// SIMATIC S7-200 project (STEP 7-Micro/WIN), CPU 224 REL 02.01

ORGANIZATION_BLOCK MAIN:OB1
TITLE=PROGRAM COMMENTS
BEGIN
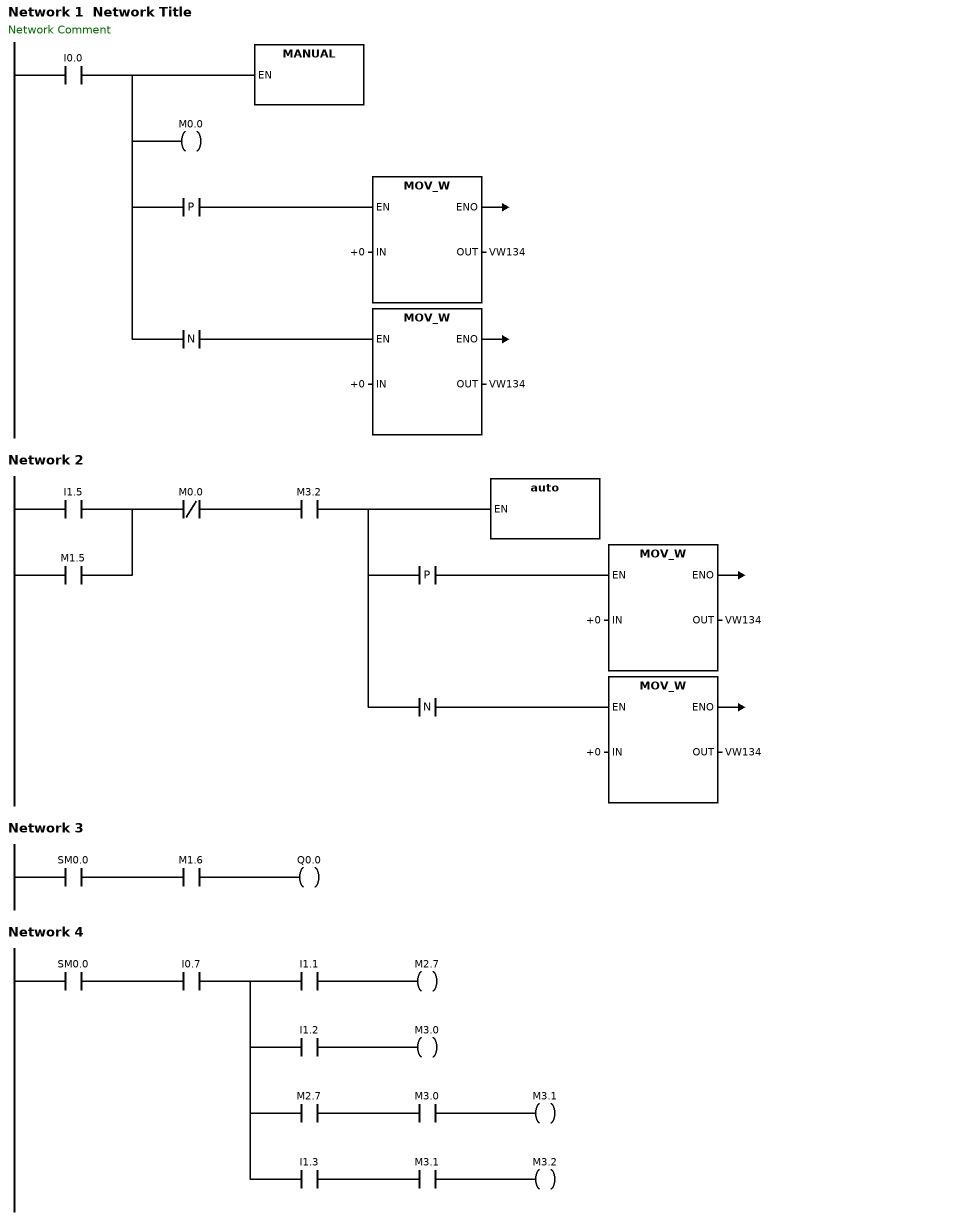
Network 1 // Network Title
// Network Comment
LD     I0.0
LPS
CALL   MANUAL:SBR0
=      M0.0
EU
MOVW   +0, VW134
LPP
ED
MOVW   +0, VW134
Network 2
LD     I1.5
O      M1.5
AN     M0.0
A      M3.2
LPS
CALL   auto:SBR1
EU
MOVW   +0, VW134
LPP
ED
MOVW   +0, VW134
Network 3
LD     SM0.0
A      M1.6
=      Q0.0
Network 4
LD     SM0.0
A      I0.7
LPS
A      I1.1
=      M2.7
LRD
A      I1.2
=      M3.0
LRD
A      M2.7
A      M3.0
=      M3.1
LPP
A      I1.3
A      M3.1
=      M3.2
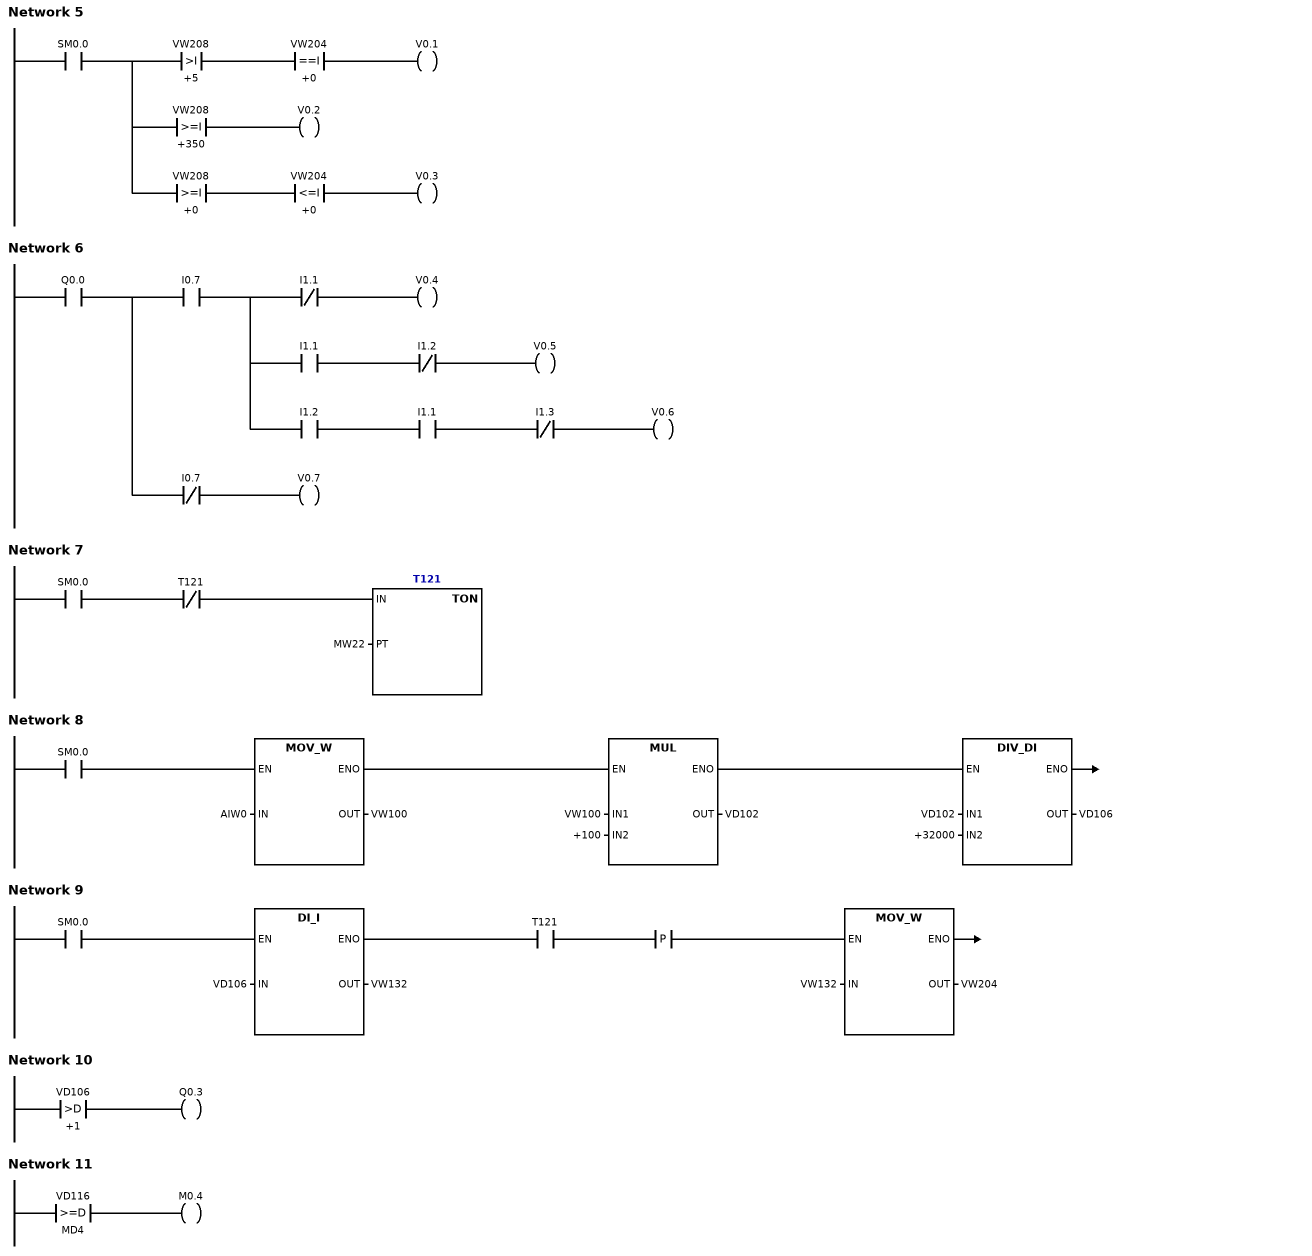
Network 5
LD     SM0.0
LPS
AW>    VW208, +5
AW=    VW204, +0
=      V0.1
LRD
AW>=   VW208, +350
=      V0.2
LPP
AW>=   VW208, +0
AW<=   VW204, +0
=      V0.3
Network 6
LD     Q0.0
LPS
A      I0.7
LPS
AN     I1.1
=      V0.4
LRD
A      I1.1
AN     I1.2
=      V0.5
LPP
A      I1.2
A      I1.1
AN     I1.3
=      V0.6
LPP
AN     I0.7
=      V0.7
Network 7
LD     SM0.0
AN     T121
TON    T121, MW22
Network 8
LD     SM0.0
MOVW   AIW0, VW100
AENO
MOVW   VW100, VW104
AENO
MUL    +100, VD102
AENO
MOVD   VD102, VD106
/D     +32000, VD106
Network 9
LD     SM0.0
DTI    VD106, VW132
AENO
A      T121
EU
MOVW   VW132, VW204
Network 10
LDD>   VD106, +1
=      Q0.3
Network 11
LDD>=  VD116, MD4
=      M0.4
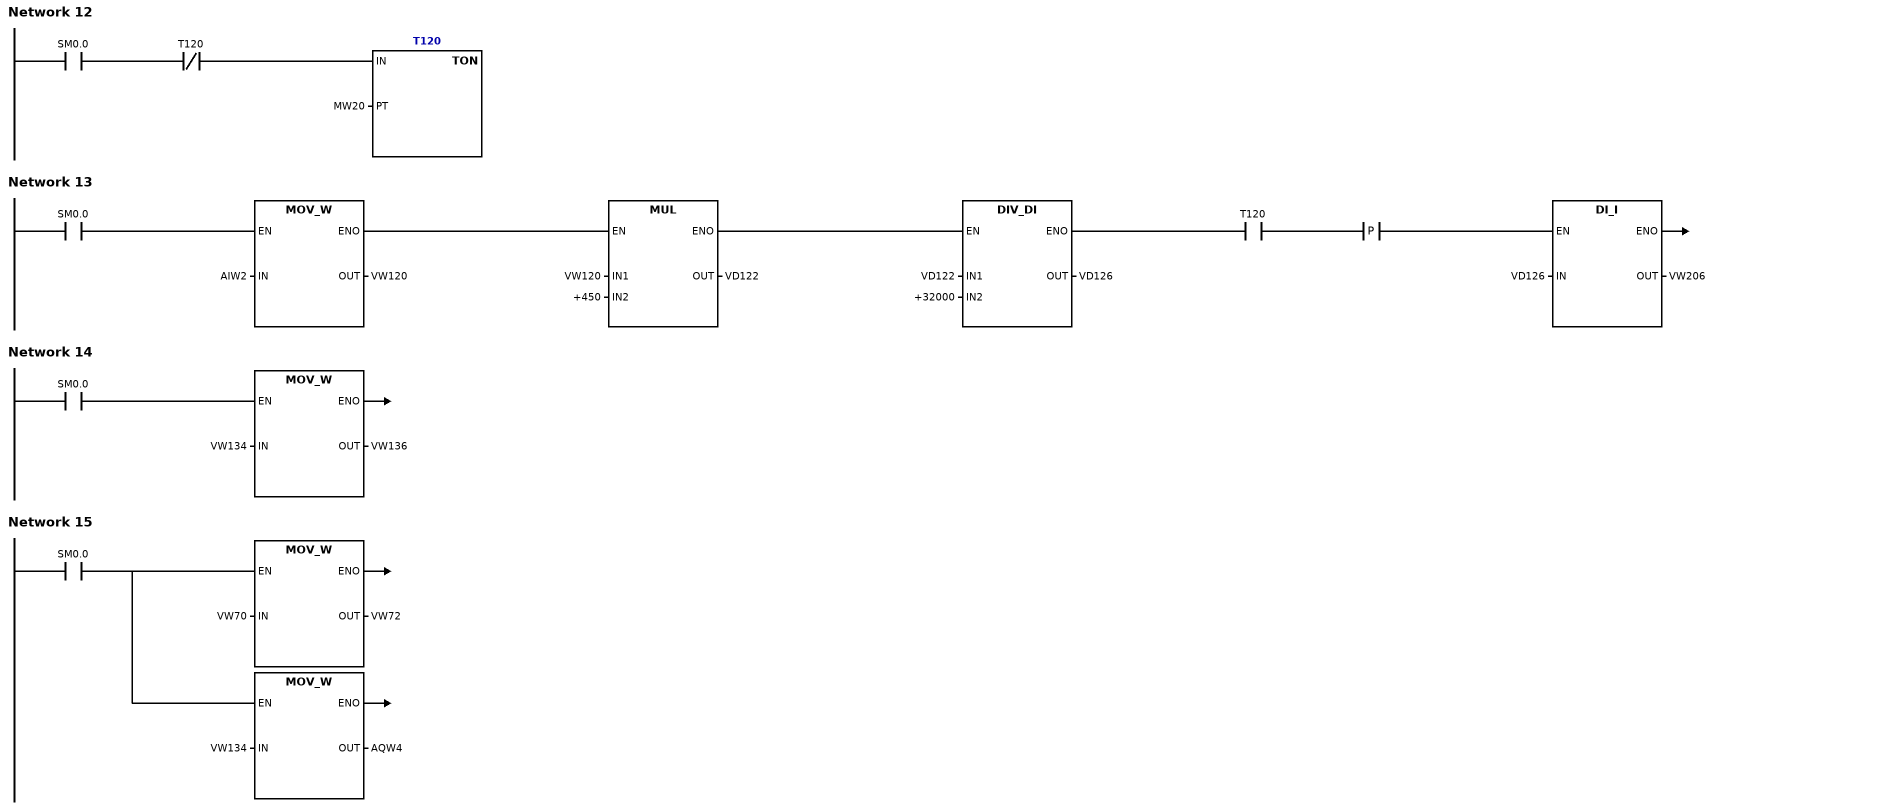
Network 12
LD     SM0.0
AN     T120
TON    T120, MW20
Network 13
LD     SM0.0
MOVW   AIW2, VW120
AENO
MOVW   VW120, VW124
AENO
MUL    +450, VD122
AENO
MOVD   VD122, VD126
AENO
/D     +32000, VD126
AENO
A      T120
EU
DTI    VD126, VW206
Network 14
LD     SM0.0
MOVW   VW134, VW136
Network 15
LD     SM0.0
MOVW   VW70, VW72
MOVW   VW134, AQW4
END_ORGANIZATION_BLOCK

SUBROUTINE_BLOCK MANUAL:SBR0
TITLE=SUBROUTINE COMMENTS
BEGIN
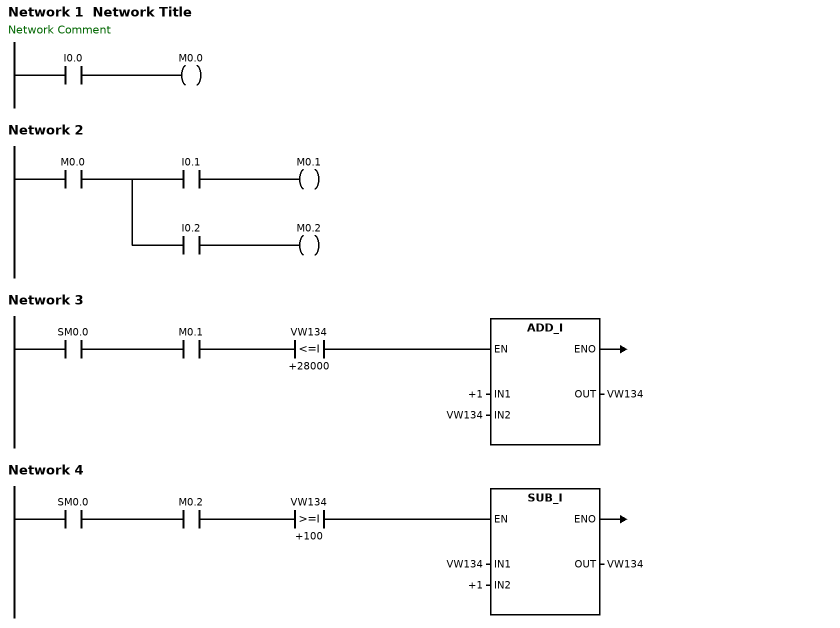
Network 1 // Network Title
// Network Comment
LD     I0.0
=      M0.0
Network 2
LD     M0.0
LPS
A      I0.1
=      M0.1
LPP
A      I0.2
=      M0.2
Network 3
LD     SM0.0
A      M0.1
AW<=   VW134, +28000
+I     +1, VW134
Network 4
LD     SM0.0
A      M0.2
AW>=   VW134, +100
-I     +1, VW134
END_SUBROUTINE_BLOCK

SUBROUTINE_BLOCK auto:SBR1
TITLE=
BEGIN
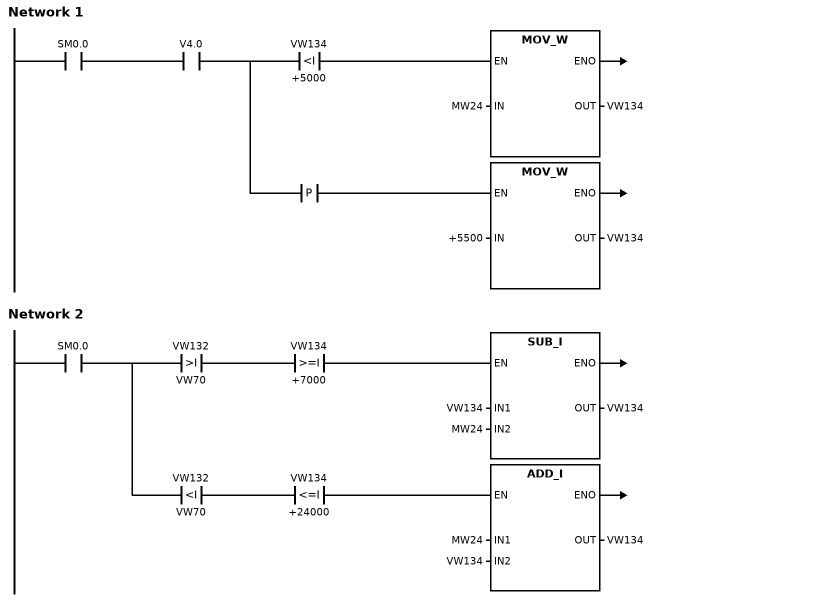
Network 1
LD     SM0.0
A      V4.0
LPS
AW<    VW134, +5000
MOVW   MW24, VW134
LPP
EU
MOVW   +5500, VW134
Network 2
LD     SM0.0
LPS
AW>    VW132, VW70
AW>=   VW134, +7000
-I     MW24, VW134
LPP
AW<    VW132, VW70
AW<=   VW134, +24000
+I     MW24, VW134
END_SUBROUTINE_BLOCK

// (further data pages could not be read)
